# EPICS IOC start-up script: jeonglee-DemoApp/iocsh/training_device.iocsh
####################################################################################################
############ START of training_device.iocsh ########################################################
#-- PREFIX         :
#-- DEVICE         :
#-- DATABASE_TOP   :
#-- PORT_NAME      :
#-- HOST           : [Default] 127.0.0.1
#-- PORT           : [Default] 9399
#-- ASYNTRACE      : [Default] ##-
#--#################################################################################################
#--#
#--#

#-- Configure the Asyn IP port using the parameters defined above
#-- drvAsynIPPortConfigure("portName", "host:port", priority, noAutoConnect, noProcessEos)
#-- priority=0 (default), noAutoConnect=0 (connect immediately), noProcessEos=0 (use Asyn default EOS processing)
drvAsynIPPortConfigure("$(PORT_NAME)", "$(HOST=127.0.0.1):$(PORT=9399)", 0, 0, 0)

#-- Configure End-of-String (EOS) terminators for the Asyn port layer
#-- These define how messages are delimited when reading from/writing to the port.
#-- Ensure these match the actual device/simulator protocol! (\n = newline, \r = carriage return)
#-- NOTE: While EOS can sometimes be defined within the StreamDevice protocol file (.proto),
#-- for long-term maintenance, it is often considered best practice to define port-specific
#-- behavior like EOS explicitly in the st.cmd file using Asyn commands.
#-- Input EOS (what character(s) mark the end of a message *received from* the device)
asynOctetSetInputEos("$(PORT_NAME)", 0, "\n")
#-- Output EOS (what character(s) should be *appended to* messages *sent to* the device)
asynOctetSetOutputEos("$(PORT_NAME)", 0, "\n")

$(ASYNTRACE=#--)asynSetTraceMask($(PORT_NAME), -1, ERROR|FLOW|DRIVER)

#-- --- Load Database Records ---
dbLoadRecords("$(DATABASE_TOP)/training.db", "P=$(PREFIX),R=$(DEVICE),PORT=$(PORT_NAME)")
#-- --- End Record Load ---

############ END of training_device.iocsh ##########################################################
####################################################################################################
